// TIA Portal V19 export
FUNCTION_BLOCK "Counter"   // FB11, LAD
{ S7_Optimized_Access := 'TRUE' }
// stored: AutoNumber false, MemoryReserve 100, SetENOAutomatically false
   VAR_INPUT
      count : Bool;
      reset : Bool;
   END_VAR
   VAR_OUTPUT
      counterValue : Int;
   END_VAR
   VAR RETAIN
      statIecCounter0 { S7_SetPoint := 'True'} : CTU_INT;
   END_VAR
BEGIN

REGION Network 1: Counter
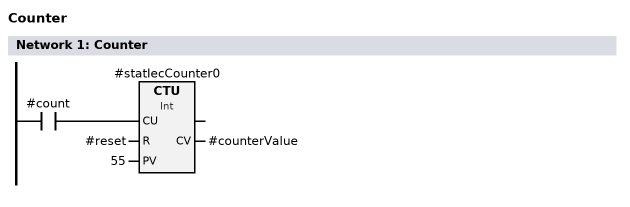
   RUNG wire#powerrail
      Contact( #count )
      { S7_Templates := "value_type := Int" } #statIecCounter0.CTU(r := #reset, pv := 55, cv => #counterValue)
   END_RUNG
   // the same network as SCL:
   #statIecCounter0(CU := #count, R := #reset, PV := 55, CV => #counterValue);   // CTU
END_REGION
END_FUNCTION_BLOCK
